(* PLC project FanoutFixture *)

PROGRAM FANOUT
  VAR  (* added by the conversion: wires and edge detectors of the diagram *)
    _OR4_OUT : BOOL;
  END_VAR

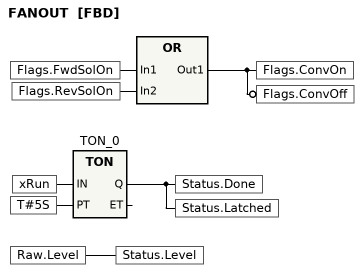
(* FBD diagram, written out as Structured Text *)
(* Conveyor off is the opposite of conveyor on *)
_OR4_OUT := Flags.FwdSolOn OR Flags.RevSolOn;
Flags.ConvOn := _OR4_OUT;
Flags.ConvOff := NOT _OR4_OUT;
(* Run timer *)
TON_0(IN := xRun, PT := T#5S);
Status.Done := TON_0.Q;
Status.Latched := TON_0.Q;
Status.Level := Raw.Level;
END_PROGRAM
